# EPICS alarm handler configuration: mps_database/bareTest/alarms/areas/mpln_bpn16_mp01.alhConfig
GROUP NULL MPLN:BPN16:MP01:1
$ALIAS MPS Link Node 80
$GUIDANCE
LTUH MPS
   Group Name: MPLN:BPN16:MP01:1
   Summary PV:  MPLN:BPN16:MP01:1:STATSUMY
$END
CHANNEL  MPLN:BPN16:MP01:1    MPLN:BPN16:MP01:1:MPS_EN_RBV		-----
CHANNEL  MPLN:BPN16:MP01:1    MPLN:BPN16:MP01:1:LC1_MODE_RBV		-----
